PROGRAM PRG_TEST
VAR
    {analysis -33}      // Disable SA0033: Unused variable
    _StringBuilder_Test : StringBuilder_Test;
END_VAR

//TcUnit.RUN();
TcUnit.RUN_IN_SEQUENCE();

END_PROGRAM

(* stored: Version 1.1.0.1
   POU PRG_TEST: Id {89d6d83b-e661-4729-8376-220f86d31845}, SpecialFunc None *)
